# EPICS substitutions: examples/test/el6022/ecmcEL6022_string.substitutions
file "ecmcEcSlave.template"
{
  pattern {}
          {}
}

file "ecmcEL6022-chX_string.template"
{
  pattern {CH_ID, PLC_ID, NELM }
          {1,     0,      22   }
          {2,     1,      22   }
}
